// TwinCAT 3 PLC project Untitled1
// ProgramVersion: 3.1.4023.0
// libraries:
//   Tc2_Standard, * (Beckhoff Automation GmbH)
//   Tc2_System, * (Beckhoff Automation GmbH)
//   Tc3_Module, * (Beckhoff Automation GmbH)
// project tree:
//   / PlcTask.TcTTO
//   POUs/ MAIN.TcPOU
// real-time tasks:
//   TASK PlcTask: cycle T#10ms, priority 20, ADS port 350
// I/O:
//   DEVICE Device 1 (CX7000), AmsNetId 5.104.86.109.2.1
//     Term 1 (CX7028) [CX7028-0000-0118]
//       modules: Module 1 (DIO_2x), Module 3 (DIO_2x), Module 5 (DI_2x), Module 7 (DI_2x)
//   DEVICE Device 2 (EtherCAT), AmsNetId 5.104.86.109.3.1
//     Term 2 (EK1200) [EK1200-5000 EtherCAT Power supply (2A E-Bus)]
//       Term 3 (EL1008) [EL1008 8Ch. Dig. Input 24V, 3ms]
//       Term 4 (EK1121-0010) [EK1121-0010 1 port EtherCAT junction (Extended Distance)]
//       Term 6 (EL9011) [EL9011 End Terminal]

CONFIGURATION Untitled1
    RESOURCE PLC ON TwinCAT3
        TASK PlcTask(INTERVAL := T#10ms, PRIORITY := 20);
        PROGRAM MAIN WITH PlcTask : MAIN;
    END_RESOURCE
END_CONFIGURATION

// ---- POUs/MAIN.TcPOU
PROGRAM MAIN
VAR
END_VAR

END_PROGRAM
